TYPE ST_FireSystem_Events_2 :
STRUCT
	CODetFault		:	BOOL;
	CODetWarning	:	BOOL;
	CODetAlarm		:	BOOL;
	SmokeDetFault	:	BOOL;
	SmokeDetAlarm	:	BOOL;
	AlarmMuted		:	BOOL;
END_STRUCT
END_TYPE

(* stored: Version 1.1.0.1, ProductVersion 3.1.4024.12
   DUT ST_FireSystem_Events_2: Id {ba64eadd-44da-409e-b2cf-6a39d668e11f} *)
